// TIA Portal V20 export
TYPE "LAxisCtrl_typeAxisConfig"
TITLE = LAxisCtrl_typeAxisConfig
// Support: tech.team.motioncontrol@siemens.com 
// Fax: +49 (0) 9131/98-1297
   STRUCT
      generalSettings { S7_SetPoint := 'True'} : "LAxisCtrl_typeGeneralSettings";   // Configuration of general settings
      power { S7_SetPoint := 'True'} : "LAxisCtrl_typePower";   // Configuration of MC_POWER function
      jog { S7_SetPoint := 'True'} : "LAxisCtrl_typeJog";   // Configuration of JOG function
      moveVelocity { S7_SetPoint := 'True'} : "LAxisCtrl_typeMoveVelocity";   // Configuration of MC_MOVEVELOCITY function
      stop { S7_SetPoint := 'True'} : "LAxisCtrl_typeStop";   // Configuration of MC_HALT function
      fastStop { S7_SetPoint := 'True'} : "LAxisCtrl_typeFastStop";   // Configuration of MC_HALT function (alternative dynamics)
      torqueLimiting { S7_SetPoint := 'True'} : "LAxisCtrl_typeTorqueLimiting";   // Configuration of MC_TORQUELIMITING function
      homing { S7_SetPoint := 'True'} : "LAxisCtrl_typeHoming";   // Configuration of HOMING function
      posRelative { S7_SetPoint := 'True'} : "LAxisCtrl_typePosRelative";   // Configuration of MC_MOVERELATIVE function
      posAbsolute { S7_SetPoint := 'True'} : "LAxisCtrl_typePosAbsolute";   // Configuration of MC_MOVEABSOLUTE function
      posSuperimposed { S7_SetPoint := 'True'} : "LAxisCtrl_typePosSuperimposed";   // Configuration of MC_MOVESUPERIMPOSED function
      gearInRelative { S7_SetPoint := 'True'} : "LAxisCtrl_typeGearInRelative";   // Configuration of MC_GEARIN function
      gearInAbsolute { S7_SetPoint := 'True'} : "LAxisCtrl_typeGearInAbsolute";   // Configuration of MC_GEARIN_POS function
      camIn { S7_SetPoint := 'True'} : "LAxisCtrl_typeCamIn";   // Configuration of MC_CAMIN function
      phasing { S7_SetPoint := 'True'} : "LAxisCtrl_typePhasing";   // Configuration of MC_PHASING function
   END_STRUCT;
END_TYPE
